(* PLC project TC3_TE1400_GeneratedModule_anarx_system_interface_FB, Beckhoff Automation GmbH & Co. KG TwinCAT 3 Function - TE1400 1.2.1240 *)
(* stored: companyURL www.beckhoff.com, creationDateTime 2022-07-14T14:06:42 *)

TYPE E_TcMatSimDataAreaType : (NotSpecified := 0, Standard, InputSrc, InputDst, OutputSrc, OutputDst, InternalDa, MArea, RetainDa);
END_TYPE

TYPE ST_TcMatSimObjectDataAreaInfo : STRUCT
  pPlcVar : PVOID;
  pModuleProcImg : PVOID;
  nSize : UDINT;
  nDataAreaId : UDINT;
  eDataAreaType : E_TcMatSimDataAreaType;
END_STRUCT;
END_TYPE

{attribute 'pack_mode' := '4'}
TYPE ST_anarx_system_interfaceInitData : STRUCT
  Header : TComInitDataHdr;
  CallByHdr : TComInitDataElmHdr;
  CallBy : TctModuleCallByType;
  ExecutionSequenceHdr : TComInitDataElmHdr;
  ExecutionSequence : TctModuleExecutionSequenceType;
  StepSizeHdr : TComInitDataElmHdr;
  StepSize : TctStepSizeType;
  ExtendedFileAccessOIDHdr : TComInitDataElmHdr;
  ExtendedFileAccessOID : OTCID;
  ExecuteModelCodeHdr : TComInitDataElmHdr;
  ExecuteModelCode : BOOL;
  ModelParametersHdr : TComInitDataElmHdr;
  ModelParameters : P_anarx_system_interface_T;
  ContextInfoArr_0_TaskOidHdr : TComInitDataElmHdr;
  ContextInfoArr_0_TaskOid : OTCID;
  ContextInfoArr_0_TaskPriorityHdr : TComInitDataElmHdr;
  ContextInfoArr_0_TaskPriority : UDINT;
  ContextInfoArr_0_TaskCycleTimeNsHdr : TComInitDataElmHdr;
  ContextInfoArr_0_TaskCycleTimeNs : UDINT;
  ContextInfoArr_0_TaskPortHdr : TComInitDataElmHdr;
  ContextInfoArr_0_TaskPort : UINT;
  ContextInfoArr_0_TaskSortOrderHdr : TComInitDataElmHdr;
  ContextInfoArr_0_TaskSortOrder : UDINT;
END_STRUCT;
END_TYPE

TYPE ST_anarx_system_interface_Input : STRUCT
  Position_Increments : UDINT;
  Velocity_Increments : LREAL;
  DMS : DINT;
  x1 : LREAL;
  y_pred : LREAL;
END_STRUCT;
END_TYPE

TYPE ST_anarx_system_interface_Output : STRUCT
  Control_Word : UINT;
  Target_Torque : INT;
  dms_kg : LREAL;
  y_anarx : LREAL;
  u_out : LREAL;
  compare_value : LREAL;
  w2 : LREAL;
  e : LREAL;
  w : LREAL;
  Out1 : BOOL;
END_STRUCT;
END_TYPE

FUNCTION_BLOCK FB_TcMatSimObject
  VAR_INPUT
    bWriteFbInputValues : BOOL := TRUE;  (* set this flag to write FB input values to the TcComObject's input DataAreas. This will overwrite the mapped input values before module execution. Set to FALSE to read the mapped input values from the TcComObject to the FB. *)
  END_VAR
  VAR
    pDataAreas : POINTER TO ST_TcMatSimObjectDataAreaInfo;  (* process image src and dst pointers and sizes *)
    nDataAreas : UDINT;
    ipObjSrv : ITComObjectServer;  (* global interface pointers *)
    ipTcComObj : ITComObject;  (* object interface pointers *)
    ipTcCyclic : ITcCyclic;
    ipTcPostCyclic : ITcPostCyclic;
    ipTcAdi : ITcADI;
    ipTask : ITcTask;  (* task interface pointers *)
    pInitData : POINTER TO TComInitDataHdr;  (* initial parameters *)
    hResult : HRESULT;  (* hResult of interface calls (0 if no error) *)
    moduleClsId : CLSID;  (* module class ID *)
    assignedClsId : CLSID;  (* expected/desired module class ID *)
    bClassIdVerified : BOOL;
    bDynInstance : BOOL;  (* flag indicating whether the module instance was created dynamically *)
    eInitialObjState : TCOM_STATE := TCOM_STATE.TCOM_STATE_INIT;  (* the object state at the time FB_init was called, FB_exit will try to switch to this state (only if this means to shift down) *)
  END_VAR

            
          

{attribute 'object_name' := 'ReleaseTcComInterface'}
METHOD ReleaseTcComInterface : HRESULT
  VAR
    nStateChangeCnt : DINT := 0;
  END_VAR
                  
IF (ipTcComObj<>0) THEN
  WHILE (State>eInitialObjState AND nStateChangeCnt<1000) DO
    State := eInitialObjState;
    nStateChangeCnt := nStateChangeCnt+1;
  END_WHILE
  ReleaseObjInterfaces();
  IF (bDynInstance) THEN
    ReleaseTcComInterface := TC3_MODULE.FW_ObjMgr_DeleteInstance(ADR(ipTcComObj));
  ELSE
    ipTcComObj.TcRelease();
  END_IF
  ipTcComObj := 0;
END_IF
                  
                
END_METHOD

{attribute 'object_name' := 'ReleaseObjInterfaces'}
METHOD ReleaseObjInterfaces : HRESULT
                  
// release interface pointers
IF (ipTcCyclic<>0) THEN
  ipTcCyclic.TcRelease();
  ipTcCyclic := 0;
END_IF
IF (ipTcPostCyclic<>0) THEN
  ipTcPostCyclic.TcRelease();
  ipTcPostCyclic := 0;
END_IF
IF (ipTcAdi<>0) THEN
  ipTcAdi.TcRelease();
  ipTcAdi := 0;
END_IF
                  
                
END_METHOD

{attribute 'object_name' := 'Internal_SetObjState'}
METHOD Internal_SetObjState
  VAR_INPUT
    hr : REFERENCE TO HRESULT;
    nextState : TCOM_STATE;
  END_VAR
                  
// verify class id
IF (SUCCEEDED(hr)) THEN
  hr := VerifyClassId();
END_IF

// switch object state
IF (SUCCEEDED(hr) AND nextState>=TCOM_STATE_INIT) THEN
  IF (ipTcComObj=0) THEN
    hr := Tc2_System.E_HRESULTAdsErr.NOINTERFACE;
  END_IF
  IF (ipObjSrv=0) THEN
    hr := Tc2_System.E_HRESULTAdsErr.NOINTERFACE;
  END_IF
  IF (SUCCEEDED(hr)) THEN
    hr := ipTcComObj.TcSetObjState(nextState,ipObjSrv,pInitData);
  END_IF
END_IF
                  
                
END_METHOD

{attribute 'object_name' := 'FB_init'}
METHOD FB_init : BOOL
  VAR_INPUT
    bInitRetains : BOOL;  (* init retain variables *)
    bInCopyCode : BOOL;  (* Online Change *)
    oid : OTCID;
  END_VAR
                  
FB_init := SUCCEEDED(Init(oid));
                  
                
END_METHOD

{attribute 'object_name' := 'GetObjPara'}
METHOD GetObjPara : HRESULT
  VAR_INPUT
    pid : PTCID;
    nData : UDINT;
    pData : PVOID;
  END_VAR
                  
IF (ipTcComObj=0) THEN
  GetObjPara := Tc2_System.E_HRESULTAdsErr.NOINTERFACE;
END_IF

IF (SUCCEEDED(GetObjPara)) THEN
  GetObjPara := ipTcComObj.TcGetObjPara(pid:=pid,nData,pData,0);
END_IF
                  
                
END_METHOD

{attribute 'object_name' := 'QueryObjInterface'}
METHOD QueryObjInterface
  VAR_INPUT
    hr : REFERENCE TO HRESULT;
    iid : REFERENCE TO IID;
    pipItf : POINTER TO ITcUnknown;
  END_VAR
  VAR CONSTANT
    pNull : PVOID := 0;
  END_VAR
                  
IF (SUCCEEDED(hr)) THEN
  IF (ipTcComObj=0) THEN
    hr := Tc2_System.E_HRESULTAdsErr.NOINTERFACE;
  ELSIF (pipItf^=ULINT_TO_DWORD(pNull)) THEN
    hr := ipTcComObj.TcQueryInterface(iid:= iid, pipItf:=pipItf);
  END_IF
END_IF
                  
                
END_METHOD

{attribute 'object_name' := 'SaveOnlineParametersForInit'}
METHOD SaveOnlineParametersForInit : HRESULT
  VAR
    idx : UINT;
    pInitElemHdr : POINTER TO TComInitDataElmHdr;
    pData : PVOID;
    nData : UDINT;
  END_VAR
  VAR CONSTANT
    nInitDataAlignment : UDINT := 4;
  END_VAR
                  IF (pInitData<>0) THEN
  pInitElemHdr := pInitData + SIZEOF(pInitData^);
  FOR idx:=1 TO pInitData^.uiElmCnt DO
    pData := pInitElemHdr + ULINT_TO_DWORD(SIZEOF(pInitElemHdr^));
    nData := pInitElemHdr^.cbData;
    SaveOnlineParametersForInit := GetObjPara(pInitElemHdr^.indexOffset,nData,pData);
    IF (FAILED(SaveOnlineParametersForInit)) THEN
      RETURN;
    END_IF
    pInitElemHdr := pData + (nInitDataAlignment*((nData + nInitDataAlignment - 1)/nInitDataAlignment));
  END_FOR
ELSE
	SaveOnlineParametersForInit := Tc2_System.E_HRESULTAdsErr.NOTINIT;
END_IF
                  
                
END_METHOD

{attribute 'object_name' := 'ResetHresult'}
METHOD ResetHresult
                  hResult := S_OK;
                
END_METHOD

{attribute 'object_name' := 'Execute'}
METHOD Execute : HRESULT
  VAR
    nDaIdx : UDINT;
    pCurDataArea : POINTER TO ST_TcMatSimObjectDataAreaInfo;
  END_VAR
                  
IF (SUCCEEDED(hResult)) THEN
  hResult := VerifyClassId();
END_IF

IF (SUCCEEDED(hResult) AND State<>TCOM_STATE_OP) THEN
  hResult := Tc2_System.E_HRESULTAdsErr.NOTREADY;
END_IF

// get image pointers
IF (SUCCEEDED(hResult)) THEN
  GetImagePtrs(hResult);
END_IF

// copy inputs
IF (pDataAreas<>0 AND nDataAreas>0 AND bWriteFbInputValues) THEN
  FOR nDaIdx:=0 TO nDataAreas-1 DO
    IF (FAILED(hResult))THEN
      CONTINUE;
    END_IF
    pCurDataArea := pDataAreas + nDaIdx*SIZEOF(ST_TcMatSimObjectDataAreaInfo);
    IF ((pCurDataArea^.eDataAreaType <> E_TcMatSimDataAreaType.InputDst))THEN
      CONTINUE;
    END_IF
    IF (pCurDataArea^.pModuleProcImg<>0 AND pCurDataArea^.pPlcVar<>0) THEN
      MEMCPY(pCurDataArea^.pModuleProcImg,pCurDataArea^.pPlcVar,pCurDataArea^.nSize);
    ELSE
      hResult := Tc2_System.E_HRESULTAdsErr.NOINTERFACE;
    END_IF
  END_FOR
END_IF

// call cycle update
IF (SUCCEEDED(hResult)) THEN
  IF (ipTcCyclic<>0) THEN
    hResult := ipTcCyclic.CycleUpdate(ipTask:= ipTask, ipCaller:= 0, context:= 0);
  ELSE
    hResult := Tc2_System.E_HRESULTAdsErr.NOINTERFACE;
  END_IF
END_IF

// copy outputs
IF (pDataAreas<>0 AND nDataAreas>0) THEN
  FOR nDaIdx:=0 TO nDataAreas-1 DO
    IF (FAILED(hResult))THEN
      CONTINUE;
    END_IF
    pCurDataArea := pDataAreas + nDaIdx*SIZEOF(ST_TcMatSimObjectDataAreaInfo);
    IF ((pCurDataArea^.eDataAreaType = E_TcMatSimDataAreaType.OutputSrc) OR NOT bWriteFbInputValues) THEN
      IF (pCurDataArea^.pModuleProcImg<>0 AND pCurDataArea^.pPlcVar<>0) THEN
        MEMCPY(pCurDataArea^.pPlcVar,pCurDataArea^.pModuleProcImg,pCurDataArea^.nSize);
      ELSE
        hResult := Tc2_System.E_HRESULTAdsErr.NOINTERFACE;
      END_IF
    END_IF
  END_FOR
END_IF


// call post cyclic update
IF (SUCCEEDED(hResult)) THEN
  IF (ipTcPostCyclic<>0) THEN
    hResult := ipTcPostCyclic.PostCyclicUpdate(ipTask:= 0, ipCaller:= 0, context:= 0);
  ELSE
    hResult := Tc2_System.E_HRESULTAdsErr.NOINTERFACE;
  END_IF
END_IF

ReleaseImagePtrs();

Execute := hResult;
                  
                
END_METHOD

{attribute 'object_name' := 'GetImagePtrs'}
METHOD GetImagePtrs
  VAR_INPUT
    hr : REFERENCE TO HRESULT;
  END_VAR
  VAR
    nDaIdx : UDINT;
    pCurDataArea : POINTER TO ST_TcMatSimObjectDataAreaInfo;
  END_VAR
                  
IF (ipTcAdi=0) THEN
  hr := Tc2_System.E_HRESULTAdsErr.NOINTERFACE;
END_IF
IF(State<>TCOM_STATE_OP)THEN
  hr := Tc2_System.E_HRESULTAdsErr.INVALIDSTATE;
END_IF


// get pointers to process images
IF (pDataAreas<>0 AND nDataAreas>0) THEN
  FOR nDaIdx:=0 TO nDataAreas-1 DO
    pCurDataArea := pDataAreas + nDaIdx*SIZEOF(ST_TcMatSimObjectDataAreaInfo);
    IF (FAILED(hr))THEN
      CONTINUE;
    END_IF
    IF ((pCurDataArea^.eDataAreaType <> E_TcMatSimDataAreaType.InputDst) AND (pCurDataArea^.eDataAreaType <> E_TcMatSimDataAreaType.OutputSrc))THEN
      CONTINUE;
    END_IF
    IF (pCurDataArea^.pModuleProcImg=0 AND pCurDataArea^.nSize>0) THEN
      hr := ipTcAdi.GetImagePtr(size:= pCurDataArea^.nSize , offs:=0 , adi_x:=pCurDataArea^.nDataAreaId , ppData:=ADR(pCurDataArea^.pModuleProcImg));
    END_IF
  END_FOR
END_IF

IF (FAILED(hr)) THEN
  ReleaseImagePtrs();
END_IF
                  
                
END_METHOD

{attribute 'object_name' := 'VerifyClassId'}
METHOD VerifyClassId : HRESULT
  VAR
    emptyClsId : CLSID;
  END_VAR
                  memset(ADR(emptyClsId),0,SIZEOF(emptyClsId));
IF (bClassIdVerified) THEN
  // class ID was already verified
  VerifyClassId := Tc2_System.E_HRESULTAdsErr.HRESULT_ADS_NOERROR;
ELSIF (memcmp(ADR(assignedClsId),ADR(emptyClsId),SIZEOF(assignedClsId))=0) THEN
  // skip class ID verification if no assignedClsId specified
  VerifyClassId := Tc2_System.E_HRESULTAdsErr.HRESULT_ADS_NOERROR;
ELSE
  // verify class ID
  VerifyClassId := ReadModuleClassId();

  IF (SUCCEEDED(VerifyClassId)) THEN
    IF (memcmp(ADR(assignedClsId),ADR(moduleClsId),SIZEOF(assignedClsId))<>0) THEN
     VerifyClassId := Tc2_System.E_HRESULTAdsErr.INVALIDCLSID;
    END_IF
  END_IF
  bClassIdVerified := SUCCEEDED(VerifyClassId);
END_IF
                  
                
END_METHOD

{attribute 'object_name' := 'SetObjPara'}
METHOD SetObjPara : HRESULT
  VAR_INPUT
    pid : PTCID;
    nData : UDINT;
    pData : PVOID;
  END_VAR
                  
IF (ipTcComObj=0) THEN
  SetObjPara := Tc2_System.E_HRESULTAdsErr.NOINTERFACE;
END_IF

IF (SUCCEEDED(SetObjPara)) THEN
  SetObjPara := ipTcComObj.TcSetObjPara(pid:=pid,nData,pData,0);
END_IF
                  
                
END_METHOD

{attribute 'object_name' := 'QueryTcComInterface'}
METHOD QueryTcComInterface
  VAR_INPUT
    hr : REFERENCE TO HRESULT;
    oid : OTCID;
  END_VAR
                  
IF (ipObjSrv=0) THEN
  hr := Tc2_System.E_HRESULTAdsErr.NOINTERFACE;
END_IF

IF (SUCCEEDED(hr) AND ipTcComObj=0) THEN
  bDynInstance := FALSE;
  IF(oid>0) THEN
    // query interface of existing object
    hr := ipObjSrv.TcQueryObjectInterface(oid,IID_ITComObject,ADR(ipTcComObj));
  ELSE
    // create new instance and get the object interface
    hr := ipObjSrv.TcCreateInstance(assignedClsId,IID_ITComObject,ADR(ipTcComObj));
    IF (SUCCEEDED(hr)) THEN
      bDynInstance := TRUE;
      hr := ipTcComObj.TcSetObjectId(OTCID_CreateNewId);
    END_IF
  END_IF
  IF (SUCCEEDED(hr)) THEN
    eInitialObjState := State;
  END_IF
END_IF
                  
                
END_METHOD

{attribute 'object_name' := 'ReleaseImagePtrs'}
METHOD ReleaseImagePtrs : HRESULT
  VAR
    nDaIdx : UDINT;
    pCurDataArea : POINTER TO ST_TcMatSimObjectDataAreaInfo;
  END_VAR
                  
IF (ipTcAdi=0) THEN
  ReleaseImagePtrs := Tc2_System.E_HRESULTAdsErr.NOINTERFACE;
END_IF

IF (SUCCEEDED(ReleaseImagePtrs) AND pDataAreas<>0 AND nDataAreas>0) THEN
  // release pointers to the simulink module process images
  FOR nDaIdx:=0 TO nDataAreas-1 DO
    pCurDataArea := pDataAreas + nDaIdx*SIZEOF(ST_TcMatSimObjectDataAreaInfo);

    IF (pCurDataArea^.pModuleProcImg<>0) THEN
      ipTcAdi.ReleaseImagePtr(pData:=pCurDataArea^.pModuleProcImg);
      pCurDataArea^.pModuleProcImg := 0;
    END_IF
  END_FOR
END_IF
                  
                
END_METHOD

{attribute 'object_name' := 'FB_exit'}
METHOD FB_exit : BOOL
  VAR_INPUT
    bInCopyCode : BOOL;  (* Online Change *)
  END_VAR
                  
IF (NOT bInCopyCode) THEN
  IF (ipObjSrv<>0) THEN
    ipObjSrv.TcRelease();
    ipObjSrv := 0;
  END_IF

  ReleaseTcComInterface();
END_IF
                  
                
END_METHOD

{attribute 'object_name' := 'InitObjName'}
METHOD InitObjName
  VAR_INPUT
    hr : REFERENCE TO HRESULT;
  END_VAR
  VAR
    objectName : STRING(255) := 'TcMatSimObject_PlcRtFbInstance';
    oid : OTCID;
  END_VAR
                  
IF (SUCCEEDED(hr)) THEN
  hr := ipTcComObj.TcGetObjectId(oid);
END_IF

IF (SUCCEEDED(hr) and bDynInstance) THEN
  objectName := TC2_STANDARD.CONCAT(objectName,'_');
  objectName := TC2_STANDARD.CONCAT(objectName,UDINT_TO_STRING(oid));
  hr := ipTcComObj.TcSetObjectName(ADR(objectName));
END_IF
                  
                
END_METHOD

{attribute 'object_name' := 'SetObjState'}
METHOD SetObjState : HRESULT
  VAR_INPUT
    finalState : TCOM_STATE;
  END_VAR
  VAR
    bShiftUp : BOOL;
    bShiftDown : BOOL;
    currentState : TCOM_STATE;
  END_VAR
                  
currentState := State;

bShiftUp := finalState>currentState;
bShiftDown := finalState<currentState;

// do not switch up on error
IF (FAILED(hresult)) THEN
  bShiftUp := FALSE;
END_IF
// reset existing error on switching down
IF (bShiftDown) THEN
  ResetHresult();
END_IF

// prepared state switch
CASE currentState OF
  TCOM_STATE_INIT:
    IF(bShiftUp) THEN
      QueryTcComInterface(hResult,0);
      Internal_SetObjState(hResult,TCOM_STATE.TCOM_STATE_PREOP);
      InitObjName(hResult);
    END_IF

  TCOM_STATE_PREOP:
    IF(bShiftUp) THEN
      Internal_SetObjState(hResult,TCOM_STATE.TCOM_STATE_SAFEOP);
      QueryObjInterfaces(hResult);
    ELSIF (bShiftDown) THEN
      Internal_SetObjState(hResult,TCOM_STATE.TCOM_STATE_INIT);
    END_IF

  TCOM_STATE_SAFEOP:
    IF(bShiftUp) THEN
      Internal_SetObjState(hResult,TCOM_STATE.TCOM_STATE_OP);
      QueryObjInterfaces(hResult);
    ELSIF (bShiftDown) THEN
      Internal_SetObjState(hResult,TCOM_STATE.TCOM_STATE_PREOP);
      ReleaseObjInterfaces();
    END_IF


  TCOM_STATE_OP:
    IF (bShiftDown) THEN
      Internal_SetObjState(hResult,TCOM_STATE.TCOM_STATE_SAFEOP);
    END_IF
END_CASE

SetObjState := hResult;
                  
                
END_METHOD

{attribute 'object_name' := 'QueryObjInterfaces'}
METHOD QueryObjInterfaces
  VAR_INPUT
    hr : REFERENCE TO HRESULT;
  END_VAR
                  
IF(State<TCOM_STATE_PREOP)THEN
  hr := Tc2_System.E_HRESULTAdsErr.INVALIDSTATE;
END_IF

//cyclic interface
QueryObjInterface(hr,IID_ITCCYCLIC,ADR(ipTcCyclic));
//post cyclic interface
QueryObjInterface(hr,IID_ITCPOSTCYCLIC,ADR(ipTcPostCyclic));
//adi interface
QueryObjInterface(hr,IID_ITcADI,ADR(ipTcAdi));
                  
                
END_METHOD

{attribute 'object_name' := 'Init'}
METHOD Init : HRESULT
  VAR_INPUT
    oid : OTCID;
  END_VAR
                  
// preinitialize variables
memset(ADR(moduleClsId),0,SIZEOF(moduleClsId));
bClassIdVerified := FALSE;
hResult := Tc2_System.E_HRESULTAdsErr.HRESULT_ADS_NOERROR;

// get object server
IF (ipObjSrv=0) THEN
  hResult := FW_ObjMgr_GetObjectServer(_AppInfo.ObjId,ADR(ipObjSrv));
END_IF

// try to get object interfaces
IF (SUCCEEDED(hresult)) THEN
  QueryTcComInterface(hResult,oid);
END_IF

// verify class id
IF (SUCCEEDED(hresult)) THEN
  hresult := VerifyClassId();
END_IF

// query interfaces, if the current state is higher than INIT
IF (SUCCEEDED(hresult) AND State>TCOM_STATE.TCOM_STATE_INIT) THEN
  QueryObjInterfaces(hResult);
END_IF

// return value
Init := hresult;
                  
                
END_METHOD

{attribute 'object_name' := 'ReadModuleClassId'}
METHOD ReadModuleClassId : HRESULT
  VAR
    emptyClsId : CLSID;
  END_VAR
                  memset(ADR(emptyClsId),0,SIZEOF(emptyClsId));
IF (memcmp(ADR(moduleClsId),ADR(emptyClsId),SIZEOF(moduleClsId))=0) THEN
  IF (ipTcComObj=0) THEN
    ReadModuleClassId := Tc2_System.E_HRESULTAdsErr.NOINTERFACE;
  END_IF

  //objectClsId := clsid;
  IF (SUCCEEDED(ReadModuleClassId)) THEN
    ReadModuleClassId := ipTcComObj.GetClassId(moduleClsId);
  END_IF
END_IF
                
END_METHOD

METHOD PUBLIC AssignClassId
VAR_INPUT
	clsId : CLSID;
END_VAR
                  assignedClsId := clsId;
bClassIdVerified := false;
                  
                
END_METHOD

PROPERTY Error : BOOL
GET
                    Error := FAILED(hResult);
                  
END_GET
END_PROPERTY

METHOD PUBLIC SetDataAreaInfo
VAR_INPUT
  pDataAreas: POINTER TO ST_TcMatSimObjectDataAreaInfo;
  nDataAreas: UDINT;
END_VAR
                  
THIS^.nDataAreas := nDataAreas;
THIS^.pDataAreas := pDataAreas;
                  
                
END_METHOD

METHOD PUBLIC SetInitDataInfo
VAR_INPUT
  pInitData : POINTER TO TComInitDataHdr;
END_VAR
                  this^.pInitData := pInitData;
                
END_METHOD

PROPERTY ClassId : CLSID
GET
                    hResult := ReadModuleClassId();
ClassId := moduleClsId;
                    
                  
END_GET
END_PROPERTY

PROPERTY State : TCOM_STATE
GET
  VAR
    hr : HRESULT := S_OK;
    eObjState : TCOM_STATE;
  END_VAR
                    
IF (ipTcComObj<>0) THEN
  hr := ipTcComObj.TcGetObjState(ADR(eObjState));
IF (FAILED(hr)) THEN
  eObjState := TCOM_STATE.TCOM_STATE_INIT;
END_IF
ELSE
  eObjState := TCOM_STATE.TCOM_STATE_INIT;
END_IF
State := eObjState;
                    
                  
END_GET
SET
                    SetObjState(State);
                  
END_SET
END_PROPERTY

PROPERTY ErrorCode : HRESULT
GET
                    ErrorCode := hResult;
                  
END_GET
END_PROPERTY
END_FUNCTION_BLOCK

{attribute 'TcDependOnClassFactory' := 'anarx_system_interface'}
FUNCTION_BLOCK FB_anarx_system_interface EXTENDS FB_TcMatSimObject
  VAR_INPUT
    stInput : ST_anarx_system_interface_Input;
  END_VAR
  VAR_OUTPUT
    stOutput : ST_anarx_system_interface_Output;
  END_VAR
  VAR
    stInitData : ST_anarx_system_interfaceInitData;
    arrDataAreas : ARRAY[1..2] OF ST_TcMatSimObjectDataAreaInfo;
    bParametersVerified : BOOL;
  END_VAR

            
          

{attribute 'object_name' := 'Internal_SetObjState'}
METHOD Internal_SetObjState
  VAR_INPUT
    hr : REFERENCE TO HRESULT;
    nextState : TCOM_STATE;
  END_VAR
                  
// update pointer to InitData structure
SetInitDataInfo(ADR(stInitData));
// call base method
SUPER^.Internal_SetObjState(hr,nextState);
                  
                
END_METHOD

{attribute 'object_name' := 'SaveOnlineParametersForInit'}
METHOD SaveOnlineParametersForInit : HRESULT
  VAR
    idx : UINT;
    pInitElemHdr : POINTER TO TComInitDataElmHdr;
    pData : PVOID;
    nData : UDINT;
  END_VAR
  VAR CONSTANT
    nInitDataAlignment : UDINT := 4;
  END_VAR
                  
// update pointer to InitData structure
SetInitDataInfo(ADR(stInitData));
// call base method
SaveOnlineParametersForInit := SUPER^.SaveOnlineParametersForInit();
                  
                
END_METHOD

METHOD FB_init : BOOL
  VAR_INPUT
    bInitRetains : BOOL;  (* if TRUE, the retain variables are initialized (warm start / cold start) *)
    bInCopyCode : BOOL;  (* if TRUE, the instance afterwards gets moved into the copy code (online change) *)
    oid : OTCID;
  END_VAR
  VAR
    clsId : CLSID;
  END_VAR
                  
// initialize flags
bParametersVerified := false;
                    
// set module class id for compatibility check
clsId.Data1 := 16#f204de61;
clsId.Data2 := 16#4840;
clsId.Data3 := 16#4670;
clsId.Data4[0] := 16#92;
clsId.Data4[1] := 16#cb;
clsId.Data4[2] := 16#3d;
clsId.Data4[3] := 16#72;
clsId.Data4[4] := 16#a9;
clsId.Data4[5] := 16#f4;
clsId.Data4[6] := 16#b4;
clsId.Data4[7] := 16#0f;

AssignClassId(clsId);
                    
// initialize InitData structure with default values              
stInitData.CallByHdr.indexGroup := 0;
stInitData.CallByHdr.indexOffset := 16#00000000;
stInitData.CallByHdr.cbData := SIZEOF(stInitData.CallBy);
stInitData.CallBy := TctModuleCallByType.CyclicTask;
stInitData.ExecutionSequenceHdr.indexGroup := 0;
stInitData.ExecutionSequenceHdr.indexOffset := 16#00000001;
stInitData.ExecutionSequenceHdr.cbData := SIZEOF(stInitData.ExecutionSequence);
stInitData.ExecutionSequence := TctModuleExecutionSequenceType.StateUpdateAfterOutputMapping;
stInitData.StepSizeHdr.indexGroup := 0;
stInitData.StepSizeHdr.indexOffset := 16#00000002;
stInitData.StepSizeHdr.cbData := SIZEOF(stInitData.StepSize);
stInitData.StepSize := TctStepSizeType.RequireMatchingTaskCycleTime;
stInitData.ExtendedFileAccessOIDHdr.indexGroup := 0;
stInitData.ExtendedFileAccessOIDHdr.indexOffset := 16#00000005;
stInitData.ExtendedFileAccessOIDHdr.cbData := SIZEOF(stInitData.ExtendedFileAccessOID);
stInitData.ExtendedFileAccessOID := 0;
stInitData.ExecuteModelCodeHdr.indexGroup := 0;
stInitData.ExecuteModelCodeHdr.indexOffset := 16#00000008;
stInitData.ExecuteModelCodeHdr.cbData := SIZEOF(stInitData.ExecuteModelCode);
stInitData.ExecuteModelCode := 1;
stInitData.ModelParametersHdr.indexGroup := 0;
stInitData.ModelParametersHdr.indexOffset := 16#83000000;
stInitData.ModelParametersHdr.cbData := SIZEOF(stInitData.ModelParameters);
stInitData.ModelParameters.WS_MAX_LENGTHS := -0.10000000000000001;
stInitData.ModelParameters.WS_MAX_VEL_m_s := 0.40000000000000002;
stInitData.ModelParameters.WS_MIN_LENGTHS := -0.20000000000000001;
stInitData.ModelParameters.u2_o := 34;
stInitData.ModelParameters.u2_s := 633;
stInitData.ModelParameters.y_o := -161456;
stInitData.ModelParameters.zero_poses := 3143153400;
stInitData.ModelParameters.PIDController_InitialConditionF := 0;
stInitData.ModelParameters.PIDController_InitialConditio_j := 0;
stInitData.ModelParameters.PIDController_LowerSaturationLi := -1.7976931348623157e+308;
stInitData.ModelParameters.PIDController_UpperSaturationLi := 1.7976931348623157e+308;
stInitData.ModelParameters.Switch2_Threshold := 0;
stInitData.ModelParameters.RESETconst_Value := 0;
stInitData.ModelParameters.BREAKFLAG_Value := 1;
stInitData.ModelParameters.Saturation1_UpperSat := 1;
stInitData.ModelParameters.Saturation1_LowerSat := 0;
stInitData.ModelParameters.velBREAK_FLAG_Value := 1;
stInitData.ModelParameters.Constant1_Value := -1;
stInitData.ModelParameters.Memory_InitialCondition := 0;
stInitData.ModelParameters.Saturation3_UpperSat := 1.7976931348623157e+308;
stInitData.ModelParameters.Saturation3_LowerSat := 0;
stInitData.ModelParameters.lenBREAK_FLAG_Value := 1;
stInitData.ModelParameters.Constant1_Value_d := -1;
stInitData.ModelParameters.Gain1_Gain := -1;
stInitData.ModelParameters.Saturation4_UpperSat := 1.7976931348623157e+308;
stInitData.ModelParameters.Saturation4_LowerSat := 0;
stInitData.ModelParameters.colBREAK_FLAG_Value := 0;
stInitData.ModelParameters.Constant1_Value_a := -1;
stInitData.ModelParameters.Constant1_Value_k := 600;
stInitData.ModelParameters.TorqueGAIN_Gain := 1;
stInitData.ModelParameters.m_endeff_Value := 0.14499999999999999;
stInitData.ModelParameters.delays_Value := 0.01;
stInitData.ModelParameters.Memory_InitialCondition_a := 0;
stInitData.ModelParameters.Saturation5_UpperSat := 1.7976931348623157e+308;
stInitData.ModelParameters.Saturation5_LowerSat := 0;
stInitData.ModelParameters.Saturation_UpperSat := 1;
stInitData.ModelParameters.Saturation_LowerSat := 0;
stInitData.ModelParameters.Gain_Gain := 200;
stInitData.ModelParameters.BreakValue_UpperSat := 1;
stInitData.ModelParameters.BreakValue_LowerSat := 0;
stInitData.ModelParameters.BREAKconst_Value := 6;
stInitData.ModelParameters.INITconst_Value := 0;
stInitData.ModelParameters.Delay_InitialCondition := 0;
stInitData.ModelParameters.Constant6_Value := 0.5;
stInitData.ModelParameters.Constant9_Value := 0;
stInitData.ModelParameters.Integrator1_IC := 0;
stInitData.ModelParameters.SineWave1_Amp := 0.5;
stInitData.ModelParameters.SineWave1_Bias := 0.5;
stInitData.ModelParameters.SineWave1_Freq := 0.10000000000000001;
stInitData.ModelParameters.SineWave1_Phase := 0;
stInitData.ModelParameters.TransferFcn_A[0] := -2000;
stInitData.ModelParameters.TransferFcn_A[1] := -1000000;
stInitData.ModelParameters.TransferFcn_C[0] := 0;
stInitData.ModelParameters.TransferFcn_C[1] := 1000000;
stInitData.ModelParameters.Constant8_Value := 1;
stInitData.ModelParameters.Gain3_Gain := 1763979.537837361;
stInitData.ModelParameters.dms_offset1_Value := 202000;
stInitData.ModelParameters.Constant_Value := 0;
stInitData.ModelParameters.Gain_Gain_l := 1.7363136810405658e-07;
stInitData.ModelParameters.Constant14_Value := 0;
stInitData.ModelParameters.Switch3_Threshold := 0;
stInitData.ModelParameters.Gain2_Gain := 1.7363136810405658e-07;
stInitData.ModelParameters.Constant13_Value := 1;
stInitData.ModelParameters.a2_Value := 0.39219999999999999;
stInitData.ModelParameters.b_Value := -0.56820000000000004;
stInitData.ModelParameters.a1_Value := 0.55830000000000002;
stInitData.ModelParameters.Constant12_Value := 0;
stInitData.ModelParameters.Gain6_Gain := 0.0015797788309636651;
stInitData.ModelParameters.Switch1_Threshold := 0;
stInitData.ModelParameters.Switch_Threshold := 0;
stInitData.ModelParameters.Constant4_Value := 0;
stInitData.ModelParameters.Constant11_Value := 0;
stInitData.ModelParameters.Constant5_Value := 0;
stInitData.ModelParameters.Constant7_Value := 100;
stInitData.ModelParameters.Gain5_Gain := 0;
stInitData.ModelParameters.enableBrakeTorque_FLAG_Value := 1;
stInitData.ModelParameters.dms_offset_Value := -202000;
stInitData.ModelParameters.Gain1_Gain_f := 5.6690000000000003e-07;
stInitData.ModelParameters.Constant10_Value := 0;
stInitData.ModelParameters.Constant2_Value := 1;
stInitData.ModelParameters.Constant3_Value := 0;
stInitData.ModelParameters.ZeroGain_Gain := 0;
stInitData.ModelParameters.Constant1_Value_p := 0;
stInitData.ModelParameters.Delay_DelayLength := 10000;
stInitData.ModelParameters.Memory_InitialCondition_aw := 0;
stInitData.ModelParameters.pause_measurement_Value := 1;
stInitData.ModelParameters.RESET_CurrentSetting := 0;
stInitData.ContextInfoArr_0_TaskOidHdr.indexGroup := 0;
stInitData.ContextInfoArr_0_TaskOidHdr.indexOffset := 16#03002060;
stInitData.ContextInfoArr_0_TaskOidHdr.cbData := SIZEOF(stInitData.ContextInfoArr_0_TaskOid);
stInitData.ContextInfoArr_0_TaskPriorityHdr.indexGroup := 0;
stInitData.ContextInfoArr_0_TaskPriorityHdr.indexOffset := 16#03002070;
stInitData.ContextInfoArr_0_TaskPriorityHdr.cbData := SIZEOF(stInitData.ContextInfoArr_0_TaskPriority);
stInitData.ContextInfoArr_0_TaskCycleTimeNsHdr.indexGroup := 0;
stInitData.ContextInfoArr_0_TaskCycleTimeNsHdr.indexOffset := 16#03002080;
stInitData.ContextInfoArr_0_TaskCycleTimeNsHdr.cbData := SIZEOF(stInitData.ContextInfoArr_0_TaskCycleTimeNs);
stInitData.ContextInfoArr_0_TaskPortHdr.indexGroup := 0;
stInitData.ContextInfoArr_0_TaskPortHdr.indexOffset := 16#03002090;
stInitData.ContextInfoArr_0_TaskPortHdr.cbData := SIZEOF(stInitData.ContextInfoArr_0_TaskPort);
stInitData.ContextInfoArr_0_TaskSortOrderHdr.indexGroup := 0;
stInitData.ContextInfoArr_0_TaskSortOrderHdr.indexOffset := 16#030020b0;
stInitData.ContextInfoArr_0_TaskSortOrderHdr.cbData := SIZEOF(stInitData.ContextInfoArr_0_TaskSortOrder);
stInitData.Header.cbData := SIZEOF(stInitData)-SIZEOF(stInitData.Header);
stInitData.Header.uiElmCnt := 11;


// set pointer to InitData structure
SetInitDataInfo(ADR(stInitData));

// set DataArea information
SetDataAreaInfo(ADR(arrDataAreas),2);
arrDataAreas[1].nDataAreaId := 0;
arrDataAreas[1].nSize := SIZEOF(stInput);
arrDataAreas[1].pPlcVar := ADR(stInput);
arrDataAreas[1].pModuleProcImg := 0;
arrDataAreas[1].eDataAreaType := E_TcMatSimDataAreaType.InputDst;
arrDataAreas[2].nDataAreaId := 1;
arrDataAreas[2].nSize := SIZEOF(stOutput);
arrDataAreas[2].pPlcVar := ADR(stOutput);
arrDataAreas[2].pModuleProcImg := 0;
arrDataAreas[2].eDataAreaType := E_TcMatSimDataAreaType.OutputSrc;


// initialize basic interface pointers and return
FB_init := SUCCEEDED(Init(oid));
                  
                
END_METHOD

METHOD Execute : HRESULT
                  
IF (SUCCEEDED(hResult)) THEN
  hResult := VerifyParameters();
END_IF

// update DataArea information
SetDataAreaInfo(ADR(arrDataAreas),2);
arrDataAreas[1].nDataAreaId := 0;
arrDataAreas[1].nSize := SIZEOF(stInput);
arrDataAreas[1].pPlcVar := ADR(stInput);
arrDataAreas[1].pModuleProcImg := 0;
arrDataAreas[1].eDataAreaType := E_TcMatSimDataAreaType.InputDst;
arrDataAreas[2].nDataAreaId := 1;
arrDataAreas[2].nSize := SIZEOF(stOutput);
arrDataAreas[2].pPlcVar := ADR(stOutput);
arrDataAreas[2].pModuleProcImg := 0;
arrDataAreas[2].eDataAreaType := E_TcMatSimDataAreaType.OutputSrc;

	
// call base method
Execute := SUPER^.Execute();
                  
                
END_METHOD

{attribute 'object_name' := 'VerifyParameters'}
METHOD VerifyParameters : HRESULT
  VAR
    moduleCallByParam : TctModuleCallByType;
  END_VAR
                  
IF (bParametersVerified) THEN
  VerifyParameters := Tc2_System.E_HRESULTAdsErr.HRESULT_ADS_NOERROR;
ELSE
  VerifyParameters := GetObjPara(stInitData.CallByHdr.indexOffset,SIZEOF(moduleCallByParam),ADR(moduleCallByParam));
  
  // check the "CallBy" parameter to be set to "Module"
  IF (SUCCEEDED(VerifyParameters) AND (moduleCallByParam <> TctModuleCallByType.Module)) THEN
      VerifyParameters := Tc2_System.E_HRESULTAdsErr.INVALIDPARM;
  END_IF
  
  // set the parameters verified flag
  bParametersVerified := SUCCEEDED(VerifyParameters);
END_IF
                  
                
END_METHOD

PROPERTY InitData : ST_anarx_system_interfaceInitData
GET
                    InitData := stInitData;
                  
END_GET
SET
                    stInitData := InitData;
                  
END_SET
END_PROPERTY
END_FUNCTION_BLOCK
